// TIA Portal V19 export
ORGANIZATION_BLOCK "Main"   // OB1, LAD, ProgramCycle
TITLE = "Main Program Sweep (Cycle)"
{ S7_Optimized_Access := 'TRUE' }
// stored: SetENOAutomatically false
   VAR_INPUT
      Initial_Call : Bool;   // Initial call of this OB
      Remanence : Bool;   // =True, if remanent data are available
   END_VAR
BEGIN

REGION Network 1
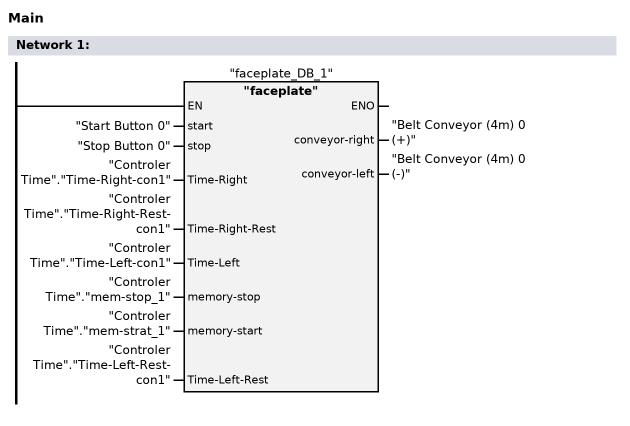
   RUNG wire#powerrail
      "faceplate_DB_1"(start := "Start Button 0", stop := "Stop Button 0", "Time-Right" := "Controler Time"."Time-Right-con1", "Time-Right-Rest" := "Controler Time"."Time-Right-Rest-con1", "Time-Left" := "Controler Time"."Time-Left-con1", "memory-stop" := "Controler Time"."mem-stop_1", "memory-start" := "Controler Time"."mem-strat_1", "Time-Left-Rest" := "Controler Time"."Time-Left-Rest-con1", "conveyor-right" => "Belt Conveyor (4m) 0 (+)", "conveyor-left" => "Belt Conveyor (4m) 0 (-)")
   END_RUNG
   // the same network as SCL:
   "faceplate_DB_1"(start := "Start Button 0",   // "faceplate"
                    stop := "Stop Button 0",
                    "Time-Right" := "Controler Time"."Time-Right-con1",
                    "Time-Right-Rest" := "Controler Time"."Time-Right-Rest-con1",
                    "Time-Left" := "Controler Time"."Time-Left-con1",
                    "memory-stop" := "Controler Time"."mem-stop_1",
                    "memory-start" := "Controler Time"."mem-strat_1",
                    "Time-Left-Rest" := "Controler Time"."Time-Left-Rest-con1",
                    "conveyor-right" => "Belt Conveyor (4m) 0 (+)",
                    "conveyor-left" => "Belt Conveyor (4m) 0 (-)");
END_REGION
END_ORGANIZATION_BLOCK
